{attribute 'linkalways'} 
{attribute 'no_explicit_call' := 'This FB is a CLASS and must be accessed using methods or properties'}
{attribute 'enable_dynamic_creation'}
FUNCTION_BLOCK _DINT EXTENDS NumericDatatypeBase
VAR
	localData : DINT;
	activeData : REFERENCE TO DINT REF= localData;
END_VAR

PROPERTY PUBLIC Address : PVOID
GET
Address := ADR(activeData);
END_GET
END_PROPERTY

METHOD PUBLIC ClearReference
VAR_INPUT
END_VAR
activeData REF= localData;
END_METHOD

METHOD PUBLIC Clone : I_Datatype
VAR
    pClone : POINTER TO _DINT;
END_VAR
pClone := __NEW(_DINT(InitialValue := Value));
Clone := pClone^;
END_METHOD

METHOD FB_init : BOOL
VAR_INPUT
	bInitRetains : BOOL; // if TRUE, the retain variables are initialized (warm start / cold start)
	bInCopyCode : BOOL;  // if TRUE, the instance afterwards gets moved into the copy code (online change)
	InitialValue : DINT;
END_VAR
localData := InitialValue;
END_METHOD

PROPERTY PUBLIC IsFloat : BOOL
GET
IsFloat := FALSE;
END_GET
END_PROPERTY

PROPERTY PUBLIC IsSigned : BOOL
GET
IsSigned := TRUE;
END_GET
END_PROPERTY

PROPERTY PUBLIC LowerBound : DINT
GET
LowerBound := DatatypeLimits.DINT_LOWER_LIMIT;
END_GET
END_PROPERTY

METHOD PUBLIC MakeReferenceTo
VAR_INPUT
	ReferenceTarget : REFERENCE TO DINT;
END_VAR
activeData REF= ReferenceTarget;
END_METHOD

PROPERTY PUBLIC Name : T_MAXSTRING
GET
Name := 'DINT';
END_GET
END_PROPERTY

METHOD PROTECTED SerializeLowerbound
VAR_INPUT
	Serializer : I_Serializer;
END_VAR
Serializer.AddDint(Lowerbound);
END_METHOD

METHOD PROTECTED SerializeUpperbound
VAR_INPUT
	Serializer : I_Serializer;
END_VAR
Serializer.AddDint(Upperbound);
END_METHOD

METHOD PUBLIC SerializeWith
VAR_INPUT
	Serializer : I_Serializer;
END_VAR
Serializer.AddDint(activeData);
END_METHOD

PROPERTY PUBLIC Size : UDINT
GET
Size := SIZEOF(activeData);
END_GET
END_PROPERTY

METHOD TryDeserializeFrom : BOOL
VAR_INPUT
	Deserializer : I_Deserializer;
	Feedback : I_DeserializerFeedback;
END_VAR
TryDeserializeFrom := Deserializer.TryGetDint(activeData, Feedback);
END_METHOD

METHOD TryMakeReferenceTo : BOOL
VAR_INPUT
	Target : I_Datatype;
END_VAR
VAR
	pTargetData : POINTER TO DINT;
END_VAR
IF NOT (Target.Name = Name) THEN
	RETURN;
END_IF

pTargetData := Target.Address;
activeData REF= pTargetData^;
TryMakeReferenceTo := TRUE;
END_METHOD

PROPERTY PUBLIC UpperBound : DINT
GET
UpperBound := DatatypeLimits.DINT_UPPER_LIMIT;
END_GET
END_PROPERTY

PROPERTY PUBLIC Value : DINT
GET
Value := activeData;
END_GET
SET
activeData := Value;
END_SET
END_PROPERTY

END_FUNCTION_BLOCK

(* stored: Version 1.1.0.1, ProductVersion 3.1.4024.12
   POU _DINT: Id {d28aeaf4-5237-00db-2a46-dbf4db665320}, SpecialFunc None
   Folder Constructor: Id {ea5562e7-14e6-054b-11e5-6d675b005757}
   Folder Protected: Id {0673644b-e5ac-0f08-236c-bdf281595d7c}
   Property Address: Id {c52b341f-d802-0a34-0a80-bac2694e1477}
   Get Get: Id {397f3b92-e865-0f79-2578-48740fab432e}
   Method ClearReference: Id {3c352e78-292a-0493-14a3-ecb6a0ba5d01}
   Method Clone: Id {a99305b5-c907-0736-22fb-797a2df46f65}
   Method FB_init: Id {7ed69fa7-a05d-0c10-2022-8ea45ef4f0c7}
   Property IsFloat: Id {48f08c8a-d026-0b99-1c24-bc7628122c99}
   Get Get: Id {1c3313e2-11ea-0e7e-00dd-527e9aefffb9}
   Property IsSigned: Id {a6b66cab-e770-0e97-21ad-c15dae53ff8d}
   Get Get: Id {4a294306-f9ec-0de8-29ca-d0cfb1c20d17}
   Property LowerBound: Id {6fc1c92c-efec-0ff5-3db1-f3aa6582d241}
   Get Get: Id {742677d1-e2af-0663-2980-c6afcdf24cc7}
   Method MakeReferenceTo: Id {762767b1-2226-0996-06f8-f6089e8950c1}
   Property Name: Id {4d666bf7-5ebf-0029-0f42-8a7f4f2344b2}
   Get Get: Id {fe4fff5d-ba25-0f2a-0a78-d1acaab61c26}
   Method SerializeLowerbound: Id {583b41c4-6632-02a4-1893-d048c2aaa795}
   Method SerializeUpperbound: Id {a9bcd55b-24b9-0785-2c7f-f9c31228740b}
   Method SerializeWith: Id {e358a02d-e70a-0fc6-07b9-b7209d612af3}
   Property Size: Id {7f06922e-b9fa-0fc3-13b7-9b78a1201719}
   Get Get: Id {866bd7da-36cd-0f2b-12ee-2d1257c759da}
   Method TryDeserializeFrom: Id {078f4f7a-3e26-0f8f-1dd5-7acc6bb4a9a4}
   Method TryMakeReferenceTo: Id {b71ac657-6c2b-0e37-3151-cfa667f3df94}
   Property UpperBound: Id {435a5257-9b41-08e2-3f3a-f000fefd93f4}
   Get Get: Id {571946c0-fda5-007e-08b8-27132446fa5c}
   Property Value: Id {febb6051-f688-0370-3e03-827527e90b18}
   Get Get: Id {5f592056-eace-0f9d-3e71-07674b9f9fb1}
   Set Set: Id {c146abec-7cc5-06ff-1c34-84d1beff35c0} *)
